(* IEC 61131-3 sources: volt/packages/volt-lsp-iec/test-corpus/lenze-mid/Device/Plc Logic/Application/MotionControl/Lenze, 9 files *)

(* ---- L_GetSlot_i700.pou ---- *)
FUNCTION L_GetSlot_i700 : INT
VAR_IN_OUT
	Axis: AXIS_REF;
END_VAR
VAR
	pAxisRef_i700: POINTER TO _AXIS_REF_i700;
END_VAR

%LANGUAGE ST
//'L_GetSlot_i700'
//
//04.2016
//Lenze Vertrieb GmbH, Mirco Guddat

(***********************************************************************************

This function check if the connected axis is an i700 axis an on witch slot it runs.
Return value:
	0 - No i700 axis
	1 - i700 axis on slot 1
	2 - i700 axis on slot 2

***********************************************************************************)

//Check if this is a i700 axis
IF (Axis.eDeviceOrigin = L_MC1P_DriveType.i700) THEN
	pAxisRef_i700:= ADR(Axis);
	IF pAxisRef_i700^.xSlot2 THEN //Check slot 2
		L_GetSlot_i700:= 2;
	ELSE
		L_GetSlot_i700:= 1;
	END_IF
ELSIF (Axis.eDeviceOrigin = L_MC1P_DriveType.i900) THEN
	L_GetSlot_i700:= 1;
ELSIF (Axis.eDeviceOrigin = L_MC1P_DriveType.i500) THEN
	L_GetSlot_i700:= 1;
ELSE
	L_GetSlot_i700:= 0; //No i700 axis
END_IF

END_FUNCTION

(* ---- ATD_FQI.pou ---- *)
FUNCTION_BLOCK ATD_FQI
VAR_INPUT
	lrAcc: LREAL:=1600;
	lrDec: LREAL:=1600;

END_VAR
VAR_OUTPUT
END_VAR
VAR
	BasicSpeed: L_MC1P_BasicActuatingSpeed;
	OffDelay: TOF;
END_VAR
VAR_IN_OUT
	ioAxis: AXIS_REF;
	DataIO: sUDT_FQIComm_Drive;;
END_VAR
%LANGUAGE LD
%NETWORK "Return when virtual axis"
ASSIGN(ioAxis.xVirtual, Q => RETURN);
%NETWORK
BasicSpeed(Axis := ioAxis, xEnableInternalControl := TRUE, xRegulatorOn := OffDelay(IN := DataIO.Controlword.Bit4_RunForward, PT := T#1S), xResetError := DataIO.Controlword.Bit7_ResetFault, xSetDriveQsp := DataIO.Controlword.Bit2_QuickStop, xEnableSetVel := DataIO.Controlword.Bit4_RunForward, xInvertDirection := DataIO.Controlword.Bit12_ReverseDirection, lrSetVel := DataIO.RefSpeed, lrSetAcc := lrAcc, lrSetDec := lrDec, xAxisReady => DataIO.Status.Bit0_ReadyForOperation, xDriveError => DataIO.Status.Bit3_Fault);

END_FUNCTION_BLOCK

(* ---- ATD_TorqueControl.pou ---- *)
FUNCTION_BLOCK ATD_TorqueControl EXTENDS ATD_FQI
VAR_INPUT
	lrTorque	: LREAL;
END_VAR
VAR_OUTPUT
END_VAR
VAR
	L_MC1P_CyclicParameterAccessWrite_0: L_MC1P_CyclicParameterAccessWrite;
END_VAR

%LANGUAGE LD
%NETWORK
SUPER^(ioAxis := ioAxis, DataIO := DataIO);
%NETWORK
L_MC1P_CyclicParameterAccessWrite_0(Axis := ioAxis, xEnable := TRUE, wIndex := 16#4008, usiSubIndex := 5, usiSize := 2, xSigned := 1, lrScaleFactor := 1, lrData := lrTorque);

END_FUNCTION_BLOCK

(* ---- BasicMovement.pou ---- *)
FUNCTION_BLOCK BasicMovement
//Dataexchange CONTROL ===========
VAR_IN_OUT
	ioDataExchange					:  sUDT_BasicMovementComm_Drive;
END_VAR
VAR_INPUT
	TouchProbeSensor				: BOOL;
	i_lrWindowStandstill			: LREAL;
	i_lrJogVel						: LREAL;
END_VAR
VAR_OUTPUT
END_VAR
VAR
	//ControlWord
	internalControl					:	BOOL;
	Control_Local			 		:	sUDT_BasicMovementComm_Drive_Control;			//output to plc

	//StatusWord

	//instance
	AxisControl						: L_TB2P_BasicMotionBase;
	SetTorqueError					: L_IE1P_SetErrorSingle;
END_VAR
VAR_IN_OUT
	ioSlaveAxis						: AXIS_REF;
END_VAR

%LANGUAGE ST

ReadInputs();
BasicMotionParameters();
BasicMotion();
SetTorqueLimits();
BrakeLogic();
WriteOutputs();

END_FUNCTION_BLOCK

METHOD BasicMotion
VAR_INPUT
END_VAR
VAR_INST
	intPositioningState		: INT;
	R_TRIG_TP				: R_TRIG;
	SetIntQspRamp			: L_SetIntQspRamp;
	lrDecErrorStopOld		: LREAL;
END_VAR
VAR

END_VAR
%LANGUAGE ST

R_TRIG_TP(CLK:=TouchProbeSensor , Q=> );

CASE intPositioningState OF
	0:	(* Wait for synchronisation *)
		AxisControl.scCtrlBasicMotion.xMoveAbsExecute := FALSE;
		AxisControl.scCtrlBasicMotion.xMoveRelExecute := FALSE;
		AxisControl.scCtrlBasicMotion.xMoveVelExecute := FALSE;
		AxisControl.scCtrlBasicMotion.xHalt := FALSE;

		IF Control_Local.StartAbsPos THEN
			intPositioningState:=10;
		ELSIF Control_Local.StartRelPos THEN
			intPositioningState:=20;
		ELSIF Control_Local.StartVelocity THEN
			intPositioningState:=30;
		ELSIF Control_Local.StartTouchprobePos THEN
			intPositioningState:=40;
		ELSIF Control_Local.StartTorqueMode THEN
			intPositioningState:=50;
		END_IF

///////////////////////////////////////////////////////////////////////////
///////////////////////////////Move absolute///////////////////////////////
///////////////////////////////////////////////////////////////////////////

	10:	(*Move absolute to position*)
		AxisControl.scPar.lrAcc := Control_Local.AccUnit;
		AxisControl.scPar.lrDec := Control_Local.DecUnit;
		AxisControl.scPar.lrVel  := Control_Local.VelUnit;
		AxisControl.scCtrlBasicMotion.lrPos_Dist := Control_Local.PosUnit;

		AxisControl.scCtrlBasicMotion.xMoveAbsExecute := TRUE;

		IF AxisControl.scStatusBasicMotion.xFunDone THEN
			ioDataExchange.Status.InPosition:=TRUE;
			intPositioningState:=15;
		ELSIF NOT Control_Local.StartAbsPos THEN
			intPositioningState:=100;
		END_IF

	15:	IF NOT Control_Local.StartAbsPos THEN
			ioDataExchange.Status.InPosition:=FALSE;
			intPositioningState:=0;
		END_IF

///////////////////////////////////////////////////////////////////////////
/////////////////////////////Move Touchprobe///////////////////////////////
///////////////////////////////////////////////////////////////////////////
	40:	(*Move Touchprobe*)
		AxisControl.scPar.lrAcc := Control_Local.AccUnit;
		AxisControl.scPar.lrDec := Control_Local.DecUnit;
		AxisControl.scPar.lrVel := Control_Local.VelUnit;

		AxisControl.scCtrlBasicMotion.xMoveVelExecute := TRUE;

		IF R_TRIG_TP.Q THEN
			AxisControl.scCtrlBasicMotion.lrPos_Dist := Control_Local.PosUnit;
			AxisControl.scCtrlBasicMotion.xMoveRelExecute := TRUE;
			intPositioningState:=41;
		ELSIF NOT Control_Local.StartTouchprobePos THEN
			intPositioningState:=100;
		END_IF

	41://wait for positioning done
		IF AxisControl.scStatusBasicMotion.xFunDone THEN
			ioDataExchange.Status.InPosition:=TRUE;
			intPositioningState:=45;
		ELSIF NOT Control_Local.StartTouchprobePos THEN
			intPositioningState:=100;
		END_IF

	45:	IF NOT Control_Local.StartTouchprobePos THEN
			ioDataExchange.Status.InPosition:=FALSE;
			intPositioningState:=0;
		END_IF

///////////////////////////////////////////////////////////////////////////
///////////////////////////////Stop movement///////////////////////////////
///////////////////////////////////////////////////////////////////////////
	100:(*Stop absolute movement*)
		AxisControl.scCtrlBasicMotion.xHalt := TRUE;

		IF AxisControl.scStatusBasicMotion.xStandstillSetVelocity THEN
			intPositioningState:=0;
		END_IF

END_CASE;

//R_TRIG_TP(CLK:=TouchProbeSensor , Q=> );

AxisControl.scCtrlBasicMotion.xResetHomePosition:=Control_Local.ResetHomePos;

AxisControl(
	xEnable:= TRUE,
	xEnableOperation:=Control_Local.Enable ,
	xResetError:=Control_Local.ResetError ,
	xQSPApplication:= ,
	xAbort:= ,
	xJogPos:= ,
	xJogNeg:= ,
	xHomeExecute:= Control_Local.ActivateHoming,
	lrOverride:= ,
	scCtrlBasicMotion:= ,
	scPar:= ,
	Axis:=ioSlaveAxis ,
	xReadyForOperation=> ,
	xOperationEnabled=> ,
	xReadyForMotion=> ,
	xError=> ,
	xWarning=> ,
	eErrorID=> ,
	xSTOActive=> ,
	xQSPActive=> ,
	xAbortBusy=> ,
	xAbortDone=> ,
	xJoggingBusy=> ,
	xHomingBusy=> ,
	xHomingDone=> ,
	xIsHomed=> ,
	eTMState=> ,
	scStatusBasicMotion=> ,
	lrActVel=> ,
	lrSetVelOut=> ,
	lrActPos=> ,
	lrSetPosOut=> ,
	lrActFollowingError=> );

SetIntQspRamp(
	Axis:=ioSlaveAxis ,
	xExecute:=ioSlaveAxis.xAxisAvailable AND NOT ioSlaveAxis.xVirtual AND (lrDecErrorStopOld=ioSlaveAxis.lrDecErrorStop) ,
	lrQspRamp:=ioSlaveAxis.lrDecErrorStop ,
	lrQspTime:= ,
	xUseQspTime:= ,
	xBusy=> ,
	xDone=> ,
	xError=> ,
	eErrorID=> );
lrDecErrorStopOld:=ioSlaveAxis.lrDecErrorStop;
END_METHOD

METHOD BasicMotionParameters
VAR_INPUT
END_VAR

%LANGUAGE ST
//General
//ioSlaveAxis.scPar.WindowStandStill:=i_lrWindowStandstill;
//ioSlaveAxis.scPar.JoggingSetVel:=i_lrJogVel;
//ioSlaveAxis.scPar.JoggingSetAcc:=i_lrJogVel*10;
//ioSlaveAxis.scPar.JoggingSetDec:=i_lrJogVel*10;
//ioSlaveAxis.scPar.JoggingSetJerk:=0;
END_METHOD

METHOD BrakeLogic
VAR_INPUT

END_VAR
VAR_INST
	BrakeInterface			: L_MC1P_BrakeInterface;
END_VAR

VAR

END_VAR
%LANGUAGE ST

BrakeInterface(
	Axis:= ioSlaveAxis,
	xEnable:= NOT ioSlaveAxis.xVirtual ,
	xReleaseBrake:= Control_Local.ReleaseBrake,
	lrTorqueAdd:= ,
	xBrakeModeActivate:= ,
	eBrakeMode:= ,
	xValid=> ,
	xBusy=> ,
	xError=> ,
	eErrorID=> ,
	xBrakeReleaseOut=> ,
	xBrakeReleased=> ,
	lrActTorque=> ,
	lrStartingTorqueSaved=> ,
	lrStartingTorqueEffective=> ,
	eBrakeModeActive=> );
END_METHOD

METHOD ReadInputs
VAR_INPUT
END_VAR

%LANGUAGE ST

//activate internal control
IF NOT internalControl THEN
	Control_Local	:= ioDataExchange.Control;
END_IF

END_METHOD

METHOD SetTorqueLimits
VAR_INPUT

END_VAR
VAR_INST
	TorqueLimit						: L_MC1P_SetTorqueLimit;
	lrRefTorqueAxis					: LREAL;
	lrActTorqueProcent				: LREAL;
	ResetError						: L_IE1P_ResetError;
END_VAR

VAR

END_VAR
%LANGUAGE ST

//Max torque on the axis. If the machine doesn't stop due to a programming error, this part ensures that the torque never gets too high.
TorqueLimit(
	Axis:= ioSlaveAxis,
	xEnable:= NOT ioSlaveAxis.xVirtual ,
	xSetTorqueLimitPos:= TRUE,
	lrTorqueLimitPos:= (Control_Local.TorqueLimit/100)*1.1, 				//The max torque allowed on the axis is 10% higher then the alarm value.
	xSetTorqueLimitNeg:= TRUE,
	lrTorqueLimitNeg:= (Control_Local.TorqueLimit/100)*1.1, 				//The max torque allowed on the axis is 10% higher then the alarm value.
	xTorqueInputAsPercent:= TRUE,
	xBusy=> ,
	xError=> ,
	eErrorID=> );

lrRefTorqueAxis := L_MC1P_GetRatedTorqueAxis(Axis:=ioSlaveAxis);
//Torque limit error
IF lrRefTorqueAxis > 0 THEN
	lrActTorqueProcent := ABS(ioSlaveAxis.lrActTorque/lrRefTorqueAxis);
END_IF

SetTorqueError(
	ModuleHandler:= ,
	ErrorHandler:=ioSlaveAxis ,
	xSetError:=lrActTorqueProcent > (Control_Local.TorqueLimit/100) ,
	eSeverity:=L_IE1P_SeverityLevel.Fault_QspAppl ,
	wTextRefId:= ATD_Errorlist,
	wErrorId:= 1,
	eReaction:= ,
	eGroup:= ,
	xError=> ,
	eErrorID=> ,
	scErrorInformation=> );

ResetError(
	ModuleHandler:= ,
	ErrorHandler:=ioSlaveAxis ,
	xResetError:=AxisControl.xResetError ,
	xError=> ,
	eErrorID=> ,
	xErrorResetActive=> ,
	xResetActive=> );
END_METHOD

METHOD WriteOutputs
VAR_INPUT
END_VAR
VAR_INST

END_VAR

%LANGUAGE ST

ioDataExchange.Status.DriveCommAlive				:= ioSlaveAxis.xCommunicationOK;
ioDataExchange.Status.ReadyForOperation				:= AxisControl.xReadyForOperation;
ioDataExchange.Status.ReadyForMotion				:= AxisControl.xReadyForMotion;
ioDataExchange.Status.HomingPosOK					:= AxisControl.xIsHomed;
ioDataExchange.Status.InPosition					;//writen in statemachine
ioDataExchange.Status.VelocitySetpointReached		;//writen in statemachine
ioDataExchange.Status.ActSpeed						:= AxisControl.lrActVel;
ioDataExchange.Status.ActPos						:= AxisControl.lrActPos;

END_METHOD

(* ---- Camming.pou ---- *)
FUNCTION_BLOCK Camming
//Dataexchange CONTROL ===========
VAR_IN_OUT
	ioDataExchange					:  sUDT_ServoComm_Drive;
END_VAR
VAR_INPUT

	i_xOnlyPositiveDirectionSync	: BOOL;
	i_lrWindowStandstill			: LREAL;
	i_lrJogVel						: LREAL;
	i_lrSyncVel 					: LREAL;
	i_NormalCamRefTable				: MC_CAM_REF;
	i_ByPassCamRefTable				: MC_CAM_REF;
	i_CamCyclic						: BOOL;
	i_MasterAbsolute				: BOOL;
	i_SlaveAbsolute					: BOOL;
END_VAR
VAR
	//ControlWord
	internalControl					:	BOOL;
	Control_Local			 		:	sUDT_ServoComm_Drive_Control;			//output to plc

	//StatusWord

	//instance
	AxisControl						: L_TS2P_FlexCamState;
	SetTorqueError					: L_IE1P_SetErrorSingle;
END_VAR
VAR_IN_OUT
	ioMasterAxis					: AXIS_REF;
	ioSlaveAxis						: AXIS_REF;
END_VAR

%LANGUAGE ST

ReadInputs();
FlexCamParameters();
FlexCam();
SetTorqueLimits();
BrakeLogic();
WriteOutputs();

END_FUNCTION_BLOCK

METHOD BrakeLogic
VAR_INPUT

END_VAR
VAR_INST
	BrakeInterface			: L_MC1P_BrakeInterface;
END_VAR

VAR

END_VAR
%LANGUAGE ST

BrakeInterface(
	Axis:= ioSlaveAxis,
	xEnable:= NOT ioSlaveAxis.xVirtual ,
	xReleaseBrake:= Control_Local.ReleaseBrake,
	lrTorqueAdd:= ,
	xBrakeModeActivate:= ,
	eBrakeMode:= ,
	xValid=> ,
	xBusy=> ,
	xError=> ,
	eErrorID=> ,
	xBrakeReleaseOut=> ,
	xBrakeReleased=> ,
	lrActTorque=> ,
	lrStartingTorqueSaved=> ,
	lrStartingTorqueEffective=> ,
	eBrakeModeActive=> );
END_METHOD

METHOD FlexCam
VAR_INPUT
END_VAR

VAR_INST
	lrMasterPos				: LREAL;
	lrSlavePos				: LREAL;
	lrDifferenceCalc		: LREAL;
	intSyncState			: INT;

	uiSetCamTable			: UINT;
	itfActiveCamTable		: MC_CAM_REF;
	CamGetSlavePosition		: L_MC2P_CamGetSlavePosition;
	xSyncCam				: BOOL;
	DelayHomePosReset	: TON;

	SetIntQspRamp			: L_SetIntQspRamp;
	lrDecErrorStopOld		: LREAL;
END_VAR
VAR

END_VAR
%LANGUAGE ST
//Selection of the cam.
IF Control_Local.SelectBypassCAM THEN
	uiSetCamTable := 2;					//Camtable 2 is a zero curve.
	itfActiveCamTable := i_ByPassCamRefTable;
ELSE
	uiSetCamTable := 1;					//Camtable 1 is the normal curve.
	itfActiveCamTable := i_NormalCamRefTable;
END_IF

//Settings for only positive synchronisation direction
IF i_xOnlyPositiveDirectionSync = TRUE AND i_SlaveAbsolute THEN

	//Get master position
	lrMasterPos := ((ioMasterAxis.lrSetPosition * AxisControl.lrSetScalingX) + AxisControl.lrSetOffsetPosX);
	IF ioMasterAxis.eTraversingRange = L_MC1P_TRAVERSINGRANGE.Modulo THEN
		lrMasterPos := L_MC1P_ModuloCycle(lrMasterPos, ioMasterAxis.lrCycleLength);
	END_IF

	//Get slave position
	CamGetSlavePosition(
		xExecute:= Control_Local.ActivateCamming,
		lrMasterPosition:= lrMasterPos,
		itfCamTable:= itfActiveCamTable,
		xDone=> ,
		xBusy=> ,
		xError=> ,
		eErrorID=> ,
		lrSlavePosition=> );
	lrSlavePos := ((CamGetSlavePosition.lrSlavePosition * AxisControl.lrSetScalingY) + AxisControl.lrSetOffsetPosY);
	IF ioSlaveAxis.eTraversingRange = L_MC1P_TRAVERSINGRANGE.Modulo THEN
		lrSlavePos := L_MC1P_ModuloCycle(lrSlavePos, ioSlaveAxis.lrCycleLength);
	END_IF

	//Calculate position difference between master and slave
	lrDifferenceCalc := L_MC1P_HlpModuloDiff(
					lrDiff:= (ioSlaveAxis.lrSetPosition - lrSlavePos),
					lrLen := ioSlaveAxis.lrCycleLength);

	//Start synchronisation
	IF ABS(lrDifferenceCalc) < 0.2 THEN
		AxisControl.scPar.eDirection := MC_DIRECTION.mcShortestWay;
	ELSE
		AxisControl.scPar.eDirection := MC_DIRECTION.mcPositiveDirection;
	END_IF

	IF NOT AxisControl.xReadyForMotion AND intSyncState>0 THEN
		intSyncState:=0;
	END_IF

	CASE intSyncState OF
		0:	(* Wait for synchronisation *)
			xSyncCam := FALSE;
			AxisControl.scCtrlBasicMotion.xMoveAbsExecute := FALSE;
			AxisControl.scCtrlBasicMotion.xHalt:=FALSE;
			AxisControl.xQSPApplication:=FALSE;

			IF Control_Local.ActivateCamming AND AxisControl.xReadyForMotion THEN
				intSyncState := 1;
			END_IF

		1:	(*Move absolute to position*)
			AxisControl.scCtrlBasicMotion.lrPos_Dist := lrSlavePos;
			AxisControl.scPar.lrAcc := AxisControl.scPar.lrSyncAcc;
			AxisControl.scPar.lrDec := AxisControl.scPar.lrSyncDec;
			AxisControl.scPar.lrVel  := AxisControl.scPar.lrSyncVel;

			AxisControl.scCtrlBasicMotion.xMoveAbsExecute := Control_Local.ActivateCamming AND CamGetSlavePosition.xDone;

			IF Control_Local.ActivateCamming = FALSE THEN
				intSyncState := 2;
			ELSIF AxisControl.scStatusBasicMotion.xFunDone = TRUE THEN
				intSyncState := 3;
			END_IF

		2:	(*Stop absolute movement*)
			AxisControl.scCtrlBasicMotion.xMoveAbsExecute := FALSE;
			AxisControl.scCtrlBasicMotion.xHalt:=TRUE;

			IF AxisControl.scStatusBasicMotion.xFunDone = TRUE THEN
				intSyncState := 0;
			END_IF

		3:	(*Synchronise drive*)
			xSyncCam := TRUE;

			IF Control_Local.ActivateCamming = FALSE THEN
				AxisControl.xQSPApplication:=TRUE;
				intSyncState := 4;
			END_IF

		4:	IF ioSlaveAxis.xStandstillSetVelocity THEN
				AxisControl.xQSPApplication:=FALSE;
				intSyncState := 0;
			END_IF

	END_CASE;
ELSE
	xSyncCam := Control_Local.ActivateCamming;
END_IF

AxisControl.scCtrlBasicMotion.xResetHomePosition:=Control_Local.ResetHomePos;

 DelayHomePosReset(IN:= NOT AxisControl.xIsHomed, PT:=T#10MS);

AxisControl(
	xEnable:=TRUE ,
	xEnableOperation:= Control_Local.Enable,
	xResetError:= Control_Local.ResetError,
	xQSPApplication:=  ,
	xAbort:=,
	xJogPos:= ,
	xJogNeg:= ,
	xHomeExecute:= Control_Local.SetHomePos AND DelayHomePosReset.q,
	lrOverride:= ,
	scCtrlBasicMotion:= ,
	scPar:= ,
	Axis:= ioSlaveAxis,
	scAccessPoints:= ,
	MasterValues:= ioMasterAxis,
	xSyncIn:= xSyncCam ,
	xCamChangeInstant:= ,
	lrSetOffsetPosX:= Control_Local.XOffset,
	lrSetOffsetPosY:= Control_Local.YOffset,
	lrSetScalingX:= ,
	lrSetScalingY:= Control_Local.YScale/1000,
	CamTable1:= i_NormalCamRefTable,
	CamTable2:= i_ByPassCamRefTable,
	CamTable3:= ,
	CamTable4:= ,
	wSetCamTable:= uiSetCamTable,
	xCamSequencer:= ,
	xReadyForOperation=> ,
	xOperationEnabled=> ,
	xReadyForMotion=> ,
	xError=> ,
	xWarning=> ,
	eErrorID=>  ,
	xSTOActive=> ,
	xQSPActive=> ,
	xAbortBusy=> ,
	xAbortDone=> ,
	xJoggingBusy=> ,
	xHomingBusy=> ,
	xHomingDone=> ,
	xIsHomed=> ,
	eTMState=> ,
	scStatusBasicMotion=> ,
	lrActVel=> ,
	lrSetVelOut=> ,
	lrActPos=> ,
	lrSetPosOut=> ,
	lrActFollowingError=> ,
	scSignalFlow=> ,
	xSynchronised=> ,
	xAccDecSync=> ,
	xCammingBusy=> ,
	xEndOfProfile=> ,
	lrOffsetPosX=> ,
	lrOffsetPosY=> ,
	wActiveCamTable=> ,
	xCamSequencerActive=> );

SetIntQspRamp(
	Axis:=ioSlaveAxis ,
	xExecute:=ioSlaveAxis.xAxisAvailable AND NOT ioSlaveAxis.xVirtual AND (lrDecErrorStopOld=ioSlaveAxis.lrDecErrorStop) ,
	lrQspRamp:=ioSlaveAxis.lrDecErrorStop ,
	lrQspTime:= ,
	xUseQspTime:= ,
	xBusy=> ,
	xDone=> ,
	xError=> ,
	eErrorID=> );
lrDecErrorStopOld:=ioSlaveAxis.lrDecErrorStop;
END_METHOD

METHOD FlexCamParameters
VAR_INPUT
END_VAR

%LANGUAGE ST
//General
//ioSlaveAxis.scPar.WindowStandStill:=i_lrWindowStandstill;
//ioSlaveAxis.scPar.JoggingSetVel:=i_lrJogVel;
//ioSlaveAxis.scPar.JoggingSetAcc:=i_lrJogVel*10;
//ioSlaveAxis.scPar.JoggingSetDec:=i_lrJogVel*10;
//ioSlaveAxis.scPar.JoggingSetJerk:=0;
//Set Flexcam Parameters
AxisControl.scPar.lrSyncVel:=i_lrSyncVel;
AxisControl.scPar.lrSyncAcc:=i_lrSyncVel*10;
AxisControl.scPar.lrSyncDec:=i_lrSyncVel*10;
AxisControl.scPar.lrSyncJerk:=0;//i_lrSyncVel*100;

AxisControl.scPar.lrSetOffsetScalingXVel:=i_lrSyncVel;
AxisControl.scPar.lrSetOffsetScalingXAcc:=i_lrSyncVel*10;
AxisControl.scPar.lrSetOffsetScalingXDec:=i_lrSyncVel*10;
AxisControl.scPar.lrSetOffsetScalingXJerk:=0;//i_lrSyncVel*100;

AxisControl.scPar.lrSetOffsetScalingYVel:=i_lrSyncVel;
AxisControl.scPar.lrSetOffsetScalingYAcc:=i_lrSyncVel*10;
AxisControl.scPar.lrSetOffsetScalingYDec:=i_lrSyncVel*10;
AxisControl.scPar.lrSetOffsetScalingYJerk:=0;//i_lrSyncVel*100;

AxisControl.scPar.eOffsetModeX:=L_TS2P_OffsetMode.ProfGenAbsolute;
AxisControl.scPar.eOffsetModeY:=L_TS2P_OffsetMode.ProfGenAbsolute;

AxisControl.scPar.eScalingModeX:=L_TS2P_ScalingMode.x_zero;
AxisControl.scPar.eScalingModeY:=L_TS2P_ScalingMode.x_zero;

AxisControl.scPar.xCamCyclic:=i_CamCyclic;
AxisControl.scPar.xMasterAbsolute:=i_MasterAbsolute;
AxisControl.scPar.xSlaveAbsolute:=i_SlaveAbsolute;

IF i_SlaveAbsolute THEN
	AxisControl.scPar.eSyncMode:=L_TS2P_SyncModeFlexCam.ProfGenAbsolute;
ELSE
	AxisControl.scPar.eSyncMode:=L_TS2P_SyncModeFlexCam.InstantRelative;
END_IF
AxisControl.scPar.lrSlaveSyncOutPos:=AxisControl.lrSetPosOut;

END_METHOD

METHOD ReadInputs
VAR_INPUT
END_VAR

%LANGUAGE ST

//activate internal control
IF NOT internalControl THEN
	Control_Local	:= ioDataExchange.Control;
END_IF

END_METHOD

METHOD SetTorqueLimits
VAR_INPUT

END_VAR
VAR_INST
	TorqueLimit						: L_MC1P_SetTorqueLimit;
	lrRefTorqueAxis					: LREAL;
	lrActTorqueProcent				: LREAL;
	ResetError						: L_IE1P_ResetError;
END_VAR

VAR

END_VAR
%LANGUAGE ST

//Max torque on the axis. If the machine doesn't stop due to a programming error, this part ensures that the torque never gets too high.
TorqueLimit(
	Axis:= ioSlaveAxis,
	xEnable:= NOT ioSlaveAxis.xVirtual ,
	xSetTorqueLimitPos:= TRUE,
	lrTorqueLimitPos:= (Control_Local.TorqueLimit/100)*1.1, 				//The max torque allowed on the axis is 10% higher then the alarm value.
	xSetTorqueLimitNeg:= TRUE,
	lrTorqueLimitNeg:= (Control_Local.TorqueLimit/100)*1.1, 				//The max torque allowed on the axis is 10% higher then the alarm value.
	xTorqueInputAsPercent:= TRUE,
	xBusy=> ,
	xError=> ,
	eErrorID=> );

lrRefTorqueAxis := L_MC1P_GetRatedTorqueAxis(Axis:=ioSlaveAxis);
//Torque limit error
IF lrRefTorqueAxis > 0 THEN
	lrActTorqueProcent := ABS(ioSlaveAxis.lrActTorque/lrRefTorqueAxis);
END_IF

SetTorqueError(
	ModuleHandler:= ,
	ErrorHandler:=ioSlaveAxis ,
	xSetError:=lrActTorqueProcent > (Control_Local.TorqueLimit/100) ,
	eSeverity:=L_IE1P_SeverityLevel.Fault_Qsp_Cinh ,
	wTextRefId:= ATD_Errorlist,
	wErrorId:= 1,
	eReaction:= ,
	eGroup:= ,
	xError=> ,
	eErrorID=> ,
	scErrorInformation=> );

ResetError(
	ModuleHandler:= ,
	ErrorHandler:=ioSlaveAxis ,
	xResetError:=AxisControl.xResetError ,
	xError=> ,
	eErrorID=> ,
	xErrorResetActive=> ,
	xResetActive=> );
END_METHOD

METHOD WriteOutputs
VAR_INPUT
END_VAR
VAR_INST

END_VAR

%LANGUAGE ST

ioDataExchange.Status.DriveCommAlive				:= ioSlaveAxis.xCommunicationOK;
ioDataExchange.Status.ReadyForOperation				:= AxisControl.xReadyForOperation;
ioDataExchange.Status.ReadyForMotion				:= AxisControl.xReadyForMotion;
ioDataExchange.Status.HomingPosOK					:= AxisControl.xIsHomed;
ioDataExchange.Status.InSync						:= AxisControl.xSynchronised;
ioDataExchange.Status.TorqueLimit					:= SetTorqueError.scErrorInformation.xError;
ioDataExchange.Status.ActSpeed						:= AxisControl.lrActVel;
ioDataExchange.Status.ActPos						:= AxisControl.lrActPos;

END_METHOD

(* ---- Camming_SideCorrection.pou ---- *)
FUNCTION_BLOCK Camming_SideCorrection EXTENDS Camming
VAR_INPUT
	i_NormalCamRefTableNeg				: MC_CAM_REF;
END_VAR
VAR_OUTPUT
END_VAR
VAR
END_VAR

%LANGUAGE ST
SUPER^( ioDataExchange:=ioDataExchange, ioMasterAxis:=ioMasterAxis,ioSlaveAxis:=ioSlaveAxis);

END_FUNCTION_BLOCK

METHOD FlexCam
VAR_INPUT
END_VAR

VAR_INST
	lrMasterPos				: LREAL;
	lrSlavePos				: LREAL;
	lrDifferenceCalc		: LREAL;
	intSyncState			: INT;

	uiSetCamTable			: UINT;
	itfActiveCamTable		: MC_CAM_REF;
	CamGetSlavePosition		: L_MC2P_CamGetSlavePosition;
	xSyncCam				: BOOL;

END_VAR
VAR

END_VAR
%LANGUAGE ST
//Selection of the cam.
IF Control_Local.SelectBypassCAM THEN
	uiSetCamTable := 2;					//Camtable 2 is a zero curve.
ELSE
	IF Control_Local.YScale<0 THEN
		uiSetCamTable := 3;					//Camtable 1 is the normal curve.
	ELSE
		uiSetCamTable := 1;					//Camtable 1 is the normal curve.
	END_IF
END_IF

//Settings for only positive synchronisation direction
IF i_xOnlyPositiveDirectionSync = TRUE AND i_SlaveAbsolute THEN

	//Get master position
	lrMasterPos := ((ioMasterAxis.lrSetPosition * AxisControl.lrSetScalingX) + AxisControl.lrSetOffsetPosX);
	IF ioMasterAxis.eTraversingRange = L_MC1P_TRAVERSINGRANGE.Modulo THEN
		lrMasterPos := L_MC1P_ModuloCycle(lrMasterPos, ioMasterAxis.lrCycleLength);
	END_IF

	//Get slave position
	CamGetSlavePosition(
		xExecute:= Control_Local.ActivateCamming,
		lrMasterPosition:= lrMasterPos,
		itfCamTable:= itfActiveCamTable,
		xDone=> ,
		xBusy=> ,
		xError=> ,
		eErrorID=> ,
		lrSlavePosition=> );
	lrSlavePos := ((CamGetSlavePosition.lrSlavePosition * AxisControl.lrSetScalingY) + AxisControl.lrSetOffsetPosY);
	IF ioSlaveAxis.eTraversingRange = L_MC1P_TRAVERSINGRANGE.Modulo THEN
		lrSlavePos := L_MC1P_ModuloCycle(lrSlavePos, ioSlaveAxis.lrCycleLength);
	END_IF

	//Calculate position difference between master and slave
	lrDifferenceCalc := L_MC1P_HlpModuloDiff(
					lrDiff:= (ioSlaveAxis.lrSetPosition - lrSlavePos),
					lrLen := ioSlaveAxis.lrCycleLength);

	//Start synchronisation
	IF ABS(lrDifferenceCalc) < 0.2 THEN
		AxisControl.scPar.eDirection := MC_DIRECTION.mcShortestWay;
	ELSE
		AxisControl.scPar.eDirection := MC_DIRECTION.mcPositiveDirection;
	END_IF

	IF NOT AxisControl.xReadyForMotion AND intSyncState>0 THEN
		intSyncState:=0;
	END_IF

	CASE intSyncState OF
		0:	(* Wait for synchronisation *)
			xSyncCam := FALSE;
			AxisControl.scCtrlBasicMotion.xMoveAbsExecute := FALSE;
			AxisControl.scCtrlBasicMotion.xHalt:=FALSE;

			IF Control_Local.ActivateCamming AND AxisControl.xReadyForMotion THEN
				intSyncState := 1;
			END_IF

		1:	(*Move absolute to position*)
			AxisControl.scCtrlBasicMotion.lrPos_Dist := lrSlavePos;
			AxisControl.scPar.lrAcc := AxisControl.scPar.lrSyncAcc;
			AxisControl.scPar.lrDec := AxisControl.scPar.lrSyncDec;
			AxisControl.scPar.lrVel  := AxisControl.scPar.lrSyncVel;

			AxisControl.scCtrlBasicMotion.xMoveAbsExecute := Control_Local.ActivateCamming AND CamGetSlavePosition.xDone;

			IF Control_Local.ActivateCamming = FALSE THEN
				intSyncState := 2;
			ELSIF AxisControl.scStatusBasicMotion.xFunDone = TRUE THEN
				intSyncState := 3;
			END_IF

		2:	(*Stop absolute movement*)
			AxisControl.scCtrlBasicMotion.xMoveAbsExecute := FALSE;
			AxisControl.scCtrlBasicMotion.xHalt:=TRUE;

			IF AxisControl.scStatusBasicMotion.xFunDone = TRUE THEN
				intSyncState := 0;
			END_IF

		3:	(*Synchronise drive*)
			xSyncCam := TRUE;

			IF Control_Local.ActivateCamming = FALSE THEN
				intSyncState := 0;
			END_IF

	END_CASE;
ELSE
	xSyncCam := Control_Local.ActivateCamming;
END_IF

AxisControl.scCtrlBasicMotion.xResetHomePosition:=Control_Local.ResetHomePos;

AxisControl(
	xEnable:=TRUE ,
	xEnableOperation:= Control_Local.Enable,
	xResetError:= Control_Local.ResetError,
	xQSPApplication:= ,
	xAbort:= ,
	xJogPos:= Control_Local.Spare2,
	xJogNeg:= Control_Local.Spare1,
	xHomeExecute:= Control_Local.SetHomePos,
	lrOverride:= ,
	scCtrlBasicMotion:= ,
	scPar:= ,
	Axis:= ioSlaveAxis,
	scAccessPoints:= ,
	MasterValues:= ioMasterAxis,
	xSyncIn:= xSyncCam,
	xCamChangeInstant:= ,
	lrSetOffsetPosX:= Control_Local.XOffset,
	lrSetOffsetPosY:= Control_Local.YOffset,
	lrSetScalingX:= ,
	lrSetScalingY:= ABS(Control_Local.YScale/1000),
	CamTable1:= i_NormalCamRefTable,
	CamTable2:= i_ByPassCamRefTable,
	CamTable3:= i_NormalCamRefTableNeg ,
	CamTable4:= ,
	wSetCamTable:= uiSetCamTable,
	xCamSequencer:= ,
	xReadyForOperation=> ,
	xOperationEnabled=> ,
	xReadyForMotion=> ,
	xError=> ,
	xWarning=> ,
	eErrorID=>  ,
	xSTOActive=> ,
	xQSPActive=> ,
	xAbortBusy=> ,
	xAbortDone=> ,
	xJoggingBusy=> ,
	xHomingBusy=> ,
	xHomingDone=> ,
	xIsHomed=> ,
	eTMState=> ,
	scStatusBasicMotion=> ,
	lrActVel=> ,
	lrSetVelOut=> ,
	lrActPos=> ,
	lrSetPosOut=> ,
	lrActFollowingError=> ,
	scSignalFlow=> ,
	xSynchronised=> ,
	xAccDecSync=> ,
	xCammingBusy=> ,
	xEndOfProfile=> ,
	lrOffsetPosX=> ,
	lrOffsetPosY=> ,
	wActiveCamTable=> ,
	xCamSequencerActive=> );
END_METHOD

(* ---- identPolePosition.pou ---- *)
FUNCTION_BLOCK identPolePosition
VAR_INPUT
	execute				: BOOL;
END_VAR
VAR_OUTPUT
	busy				: BOOL;
	done				: BOOL;
	doneOnce			: BOOL;
	error				: BOOL;
	polePositionOld		: LREAL;
	polePositionNew		: LREAL;
END_VAR
VAR
	iStep: INT;
	MC_ReadParameter	: MC_ReadParameter;
	MC_WriteParameter	: MC_WriteParameter;
	TON:TON;
END_VAR
VAR_IN_OUT
	ioAxis				: AXIS_REF;
END_VAR
%LANGUAGE ST

CASE iStep OF

	0:	MC_ReadParameter.Enable:=FALSE;
		MC_WriteParameter.Execute:=FALSE;
		done:=FALSE;
		busy:=FALSE;
		error:=FALSE;

		IF execute THEN
			busy:=true;
			iStep:=2;
		END_IF

	2:	//Read	0x3024:0	Device control via PDO: Activation	Activate [1]
		MC_ReadParameter.Enable:=TRUE;
		MC_ReadParameter.ParameterNumber:=L_MC1P_IndexToParameter2(
				uiIndex:=16#3024 ,
				usiSubIndex:=0 ,
				uiByteLength:=1 ,
				xUnsigned:=TRUE );

		IF MC_ReadParameter.Valid THEN
			//IF MC_ReadParameter.Value = 1 THEN
				MC_ReadParameter.Enable:=FALSE;
				iStep:=4;
			//ELSE
			//	error:=TRUE;
			//END_IF
		ELSIF NOT execute THEN
			iStep:=0;
		ELSIF MC_ReadParameter.Error THEN
			error:=TRUE;
		END_IF

	4:	//Write	0x3024:0	Device control via PDO: Activation	Off [0]
		MC_WriteParameter.Execute:=TRUE;
		MC_WriteParameter.ParameterNumber:=L_MC1P_IndexToParameter2(
				uiIndex:=16#3024 ,
				usiSubIndex:=0 ,
				uiByteLength:=1 ,
				xUnsigned:=TRUE );
		MC_WriteParameter.Value:=0;

		IF MC_WriteParameter.Done THEN
			MC_WriteParameter.Execute:=FALSE;
			iStep:=6;
		ELSIF NOT execute THEN
			iStep:=0;
		ELSIF MC_WriteParameter.Error THEN
			error:=TRUE;
		END_IF

	6:	//Read	0x3025:0	Mode: Selection	CiA402 mode active [0]
		MC_ReadParameter.Enable:=TRUE;
		MC_ReadParameter.ParameterNumber:=L_MC1P_IndexToParameter2(
				uiIndex:=16#3025 ,
				usiSubIndex:=0 ,
				uiByteLength:=1 ,
				xUnsigned:=TRUE );

		IF MC_ReadParameter.Valid THEN
			//IF MC_ReadParameter.Value = 0 THEN
				MC_ReadParameter.Enable:=FALSE;
				iStep:=8;
			//ELSE
			//	error:=TRUE;
			//END_IF
		ELSIF NOT execute THEN
			iStep:=0;
		ELSIF MC_ReadParameter.Error THEN
			error:=TRUE;
		END_IF

	8:	//Write	0x3025:0	Mode: Selection	Pole position identification PPI (without movement) [7]
		MC_WriteParameter.Execute:=TRUE;
		MC_WriteParameter.ParameterNumber:=L_MC1P_IndexToParameter2(
				uiIndex:=16#3025 ,
				usiSubIndex:=0 ,
				uiByteLength:=1 ,
				xUnsigned:=TRUE );
		MC_WriteParameter.Value:=7;

		IF MC_WriteParameter.Done THEN
			MC_WriteParameter.Execute:=FALSE;
			iStep:=10;
		ELSIF NOT execute THEN
			iStep:=0;
		ELSIF MC_WriteParameter.Error THEN
			error:=TRUE;
		END_IF

	10:	//Read	0x3403:4	Motor (SM): Pole position encoder	49,5	°
		MC_ReadParameter.Enable:=TRUE;
		MC_ReadParameter.ParameterNumber:=L_MC1P_IndexToParameter2(
				uiIndex:=16#3403 ,
				usiSubIndex:=4 ,
				uiByteLength:=2 ,
				xUnsigned:=TRUE );

		IF MC_ReadParameter.Valid THEN
			polePositionOld:=MC_ReadParameter.Value;
			MC_ReadParameter.Enable:=FALSE;
			iStep:=12;
		ELSIF NOT execute THEN
			iStep:=0;
		ELSIF MC_ReadParameter.Error THEN
			error:=TRUE;
		END_IF

	12://Write	0x6840:0	Controlword	0x0006
		MC_WriteParameter.Execute:=TRUE;
		MC_WriteParameter.ParameterNumber:=L_MC1P_IndexToParameter2(
				uiIndex:=16#6840 ,
				usiSubIndex:=0 ,
				uiByteLength:=2 ,
				xUnsigned:=TRUE );
		MC_WriteParameter.Value:=16#0006;

		IF MC_WriteParameter.Done THEN
			MC_WriteParameter.Execute:=FALSE;
			iStep:=14;
		ELSIF NOT execute THEN
			iStep:=0;
		ELSIF MC_WriteParameter.Error THEN
			error:=TRUE;
		END_IF

	14://Read	0x6841:0	Statusword	0x0021
		MC_ReadParameter.Enable:=TRUE;
		MC_ReadParameter.ParameterNumber:=L_MC1P_IndexToParameter2(
				uiIndex:=16#6841 ,
				usiSubIndex:=0 ,
				uiByteLength:=2 ,
				xUnsigned:=TRUE );

		IF MC_ReadParameter.Valid THEN
			//IF MC_ReadParameter.Value = 16#0021 THEN
				MC_ReadParameter.Enable:=FALSE;
				iStep:=16;
			//ELSE
			//	error:=TRUE;
			//END_IF
		ELSIF NOT execute THEN
			iStep:=0;
		ELSIF MC_ReadParameter.Error THEN
			error:=TRUE;
		END_IF

	16://Write	0x6840:0	Controlword	0x0007
		MC_WriteParameter.Execute:=TRUE;
		MC_WriteParameter.ParameterNumber:=L_MC1P_IndexToParameter2(
				uiIndex:=16#6840 ,
				usiSubIndex:=0 ,
				uiByteLength:=2 ,
				xUnsigned:=TRUE );
		MC_WriteParameter.Value:=16#0007;

		IF MC_WriteParameter.Done THEN
			MC_WriteParameter.Execute:=FALSE;
			iStep:=18;
		ELSIF NOT execute THEN
			iStep:=0;
		ELSIF MC_WriteParameter.Error THEN
			error:=TRUE;
		END_IF

	18://Read	0x6841:0	Statusword	0x0023
		MC_ReadParameter.Enable:=TRUE;
		MC_ReadParameter.ParameterNumber:=L_MC1P_IndexToParameter2(
				uiIndex:=16#6841 ,
				usiSubIndex:=0 ,
				uiByteLength:=2 ,
				xUnsigned:=TRUE );

		IF MC_ReadParameter.Valid THEN
			//IF MC_ReadParameter.Value = 16#0023 THEN
				MC_ReadParameter.Enable:=FALSE;
				iStep:=20;
			//ELSE
			//	error:=TRUE;
			//END_IF
		ELSIF NOT execute THEN
			iStep:=0;
		ELSIF MC_ReadParameter.Error THEN
			error:=TRUE;
		END_IF

	20://Write	0x6840:0	Controlword	0x000F
		MC_WriteParameter.Execute:=TRUE;
		MC_WriteParameter.ParameterNumber:=L_MC1P_IndexToParameter2(
				uiIndex:=16#6840 ,
				usiSubIndex:=0 ,
				uiByteLength:=2 ,
				xUnsigned:=TRUE );
		MC_WriteParameter.Value:=16#000F;

		IF MC_WriteParameter.Done THEN
			MC_WriteParameter.Execute:=FALSE;
			TON(IN:=FALSE);
			iStep:=22;
		ELSIF NOT execute THEN
			iStep:=0;
		ELSIF MC_WriteParameter.Error THEN
			error:=TRUE;
		END_IF

	22://Check for finished
		TON(IN:=TRUE , PT:= T#5S, Q=> , ET=> );

		IF TON.Q THEN
			iStep:=24;
		ELSIF NOT execute THEN
			iStep:=0;
		END_IF

	24://Write	0x6840:0	Controlword	0x0000
		MC_WriteParameter.Execute:=TRUE;
		MC_WriteParameter.ParameterNumber:=L_MC1P_IndexToParameter2(
				uiIndex:=16#6840 ,
				usiSubIndex:=0 ,
				uiByteLength:=2 ,
				xUnsigned:=TRUE );
		MC_WriteParameter.Value:=16#0000;

		IF MC_WriteParameter.Done THEN
			MC_WriteParameter.Execute:=FALSE;
			iStep:=26;
		ELSIF NOT execute THEN
			iStep:=0;
		ELSIF MC_WriteParameter.Error THEN
			error:=TRUE;
		END_IF

	26:	//Read	0x3403:4	Motor (SM): Pole position encoder	49,5	°
		MC_ReadParameter.Enable:=TRUE;
		MC_ReadParameter.ParameterNumber:=L_MC1P_IndexToParameter2(
				uiIndex:=16#3403 ,
				usiSubIndex:=4 ,
				uiByteLength:=2 ,
				xUnsigned:=TRUE );

		IF MC_ReadParameter.Valid THEN
			polePositionNew:=MC_ReadParameter.Value;
			MC_ReadParameter.Enable:=FALSE;
			iStep:=28;
		ELSIF NOT execute THEN
			iStep:=0;
		ELSIF MC_ReadParameter.Error THEN
			error:=TRUE;
		END_IF

	28://Save	0x3403:4	Motor (SM): Pole position encoder	51,7	°
		MC_WriteParameter.Execute:=TRUE;
		MC_WriteParameter.ParameterNumber:=L_MC1P_IndexToParameter2(
				uiIndex:=16#3403 ,
				usiSubIndex:=4 ,
				uiByteLength:=2 ,
				xUnsigned:=TRUE );
		MC_WriteParameter.Value:=polePositionNew;

		IF MC_WriteParameter.Done THEN
			MC_WriteParameter.Execute:=FALSE;
			iStep:=30;
		ELSIF NOT execute THEN
			iStep:=0;
		ELSIF MC_WriteParameter.Error THEN
			error:=TRUE;
		END_IF

	30:	//Write	0x3025:0	Mode: Selection	CiA402 mode active [0]
		MC_WriteParameter.Execute:=TRUE;
		MC_WriteParameter.ParameterNumber:=L_MC1P_IndexToParameter2(
				uiIndex:=16#3025 ,
				usiSubIndex:=0 ,
				uiByteLength:=1 ,
				xUnsigned:=TRUE );
		MC_WriteParameter.Value:=0;

		IF MC_WriteParameter.Done THEN
			MC_WriteParameter.Execute:=FALSE;
			iStep:=32;
		ELSIF NOT execute THEN
			iStep:=0;
		ELSIF MC_WriteParameter.Error THEN
			error:=TRUE;
		END_IF

	32:	//Write	0x3024:0	Device control via PDO: Activation	Off [0]
		MC_WriteParameter.Execute:=TRUE;
		MC_WriteParameter.ParameterNumber:=L_MC1P_IndexToParameter2(
				uiIndex:=16#3024 ,
				usiSubIndex:=0 ,
				uiByteLength:=1 ,
				xUnsigned:=TRUE );
		MC_WriteParameter.Value:=1;

		IF MC_WriteParameter.Done THEN
			MC_WriteParameter.Execute:=FALSE;
			iStep:=100;
		ELSIF NOT execute THEN
			iStep:=0;
		ELSIF MC_WriteParameter.Error THEN
			error:=TRUE;
		END_IF

	100://Pole ident done
		done:=TRUE;
		doneOnce:=TRUE;
		busy:=FALSE;
		IF NOT execute THEN
			done:=FALSE;
			iStep:=0;
		END_IF
END_CASE

MC_WriteParameter(
	Axis:=ioAxis ,
	Execute:= ,
	ParameterNumber:= ,
	Value:= ,
	ExecutionMode:= ,
	Done=> ,
	Busy=> ,
	Error=> ,
	ErrorID=> );

MC_ReadParameter(
	Axis:=ioAxis ,
	Enable:= ,
	ParameterNumber:= ,
	Valid=> ,
	Busy=> ,
	Error=> ,
	ErrorID=> ,
	Value=> );

	(*
L_ETC_CoE_SdoRead4(
	xExecute:= ,
	xAbort:= ,
	usiCom:= ,
	uiDevice:=uiDevice ,
	wIndex:= ,
	bySubindex:= ,
	udiTimeOut:=100 ,
	xDone=> ,
	xBusy=> ,
	xError=> ,
	eErrorCode=> ,
	udiSdoAbort=> ,
	abyData=> ,
	szDataRead=> );

L_ETC_CoE_SdoWrite4(
	xExecute:= ,
	xAbort:= ,
	usiCom:= ,
	uiDevice:=uiDevice ,
	wIndex:= ,
	bySubindex:= ,
	udiTimeOut:=100 ,
	abyData:= ,
	usiDataLength:= ,
	xDone=> ,
	xBusy=> ,
	xError=> ,
	eErrorCode=> ,
	udiSdoAbort=> );
*)

END_FUNCTION_BLOCK

(* ---- L_SetIntQspRamp.pou ---- *)
FUNCTION_BLOCK L_SetIntQspRamp
VAR_IN_OUT
	Axis: AXIS_REF;
END_VAR
VAR_INPUT
	xExecute: BOOL;
	lrQspRamp: LREAL;
	lrQspTime: LREAL;
	xUseQspTime: BOOL;
END_VAR
VAR_OUTPUT
	xBusy: BOOL;
	xDone: BOOL;
	xError: BOOL;
	eErrorID: L_IE1P_Error;
END_VAR
VAR
	L_MC1P_ReadMachineData_Axis: L_MC1P_ReadMachineData;
	MC_WriteParameter_QspRamp: MC_WriteParameter;
	lrQspRamp_PosUnit: LREAL;
	RatedVel: LREAL;
	iStep: INT;
	uiIndexQspRamp: UINT;
	iSlotAxis: INT;
END_VAR

%LANGUAGE ST
//'L_SetIntQspRamp_i700'
//
//04.2016
//Lenze Vertrieb GmbH, Mirco Guddat

//Check if this is a i700 axis and witch slot
iSlotAxis:= L_GetSlot_i700(Axis:= Axis);

CASE iStep OF
	0: //Start
		xDone:= FALSE;
		xBusy:= FALSE;
		MC_WriteParameter_QspRamp.Execute:= FALSE;
		L_MC1P_ReadMachineData_Axis.xEnable:= FALSE;
		xError:= FALSE;
		eErrorID:= L_IE1P_Error.NoError;

		IF xExecute THEN
			iStep:= 10;
		END_IF

	10: //Read machine data
		xBusy:= TRUE;
		L_MC1P_ReadMachineData_Axis.xEnable:= TRUE;

		IF L_MC1P_ReadMachineData_Axis.xValid THEN
			iStep:= 20;
			ELSIF L_MC1P_ReadMachineData_Axis.xError THEN
				xError:= TRUE;
				eErrorID:= L_MC1P_ReadMachineData_Axis.eErrorID;
				iStep:= 40;
		END_IF

	20: //Calculate the internal quickstop ramp in Pos.Units/s2
		IF xUseQspTime THEN

			IF lrQspTime> 0 THEN
				IF (L_MC1P_ReadMachineData_Axis.lrFeedconstant= 0) OR (L_MC1P_ReadMachineData_Axis.dwGearDenominator= 0) THEN
					//Division by zero
					xError:= TRUE;
					lrQspRamp_PosUnit:= 16#7FFFFFFF;

					ELSE
						//The QSP-Time is calculated from rated velocity to standstill
						lrQspRamp_PosUnit:= ((L_MC1P_GetRatedVelocityAxis(Axis:= Axis)/ L_MC1P_ReadMachineData_Axis.lrFeedconstant) * (TO_LREAL(L_MC1P_ReadMachineData_Axis.dwGearNumerator) / TO_LREAL(L_MC1P_ReadMachineData_Axis.dwGearDenominator)) / lrQspTime) * 65536;
				END_IF

				ELSE
					//Zero dont work as QSP time, so we use the max. deceleration
					lrQspRamp_PosUnit:= 16#7FFFFFFF;
			END_IF

			ELSE
				IF lrQspRamp> 0.0 THEN
					IF (L_MC1P_ReadMachineData_Axis.lrFeedconstant= 0) OR (L_MC1P_ReadMachineData_Axis.dwGearDenominator= 0) THEN
						//Division by zero
						xError:= TRUE;
						lrQspRamp_PosUnit:= 16#7FFFFFFF;

						ELSE
							//Calculate QSP ramp
							lrQspRamp_PosUnit:= (lrQspRamp/ L_MC1P_ReadMachineData_Axis.lrFeedconstant) * (TO_LREAL(L_MC1P_ReadMachineData_Axis.dwGearNumerator) / TO_LREAL(L_MC1P_ReadMachineData_Axis.dwGearDenominator)) * 65536;
					END_IF

					ELSE
						//Zero dont work as QSP ramp, so we use the max. deceleration
						lrQspRamp_PosUnit:= 16#7FFFFFFF;
				END_IF
		END_IF

		iStep:= 30;

	30: //Write the parameter
		IF (iSlotAxis= 1) THEN
			uiIndexQspRamp:= 16#6085; //Index for slot 1
			ELSIF (iSlotAxis= 2) THEN
				uiIndexQspRamp:= 16#6885; //Index for slot 2
		END_IF

		MC_WriteParameter_QspRamp.Execute:= TRUE;

		IF MC_WriteParameter_QspRamp.Done THEN
			iStep:= 40;
			ELSIF MC_WriteParameter_QspRamp.Error THEN
				xError:= TRUE;
				eErrorID:= MC_WriteParameter_QspRamp.ErrorID;
		END_IF

	40: //finish
		xDone:= TRUE;
		xBusy:= FALSE;
		IF NOT xExecute THEN
			iStep:= 0;
		END_IF

END_CASE

L_MC1P_ReadMachineData_Axis(
	Axis:= Axis,
	xEnable:= ,
	xValid=> ,
	xBusy=> ,
	xError=> ,
	eErrorID=> ,
	lrFeedconstant=> ,
	dwGearDenominator=> ,
	dwGearNumerator=> ,
	dwPosResolution=> ,
	xOrientation=> ,
	eTraversingRange=> ,
	lrCycleLength=> ,
	xVirtual=> );

MC_WriteParameter_QspRamp(
	Axis:= Axis,
	Execute:= ,
	ParameterNumber:= L_MC1P_IndexToParameter(uiIndex:= uiIndexQspRamp, usiSubIndex:= 0, uiByteLength:= 4),
	Value:= lrQspRamp_PosUnit,
	ExecutionMode:= ,
	Done=> ,
	Busy=> ,
	Error=> ,
	ErrorID=> );

END_FUNCTION_BLOCK

(* ---- VirtualMaster.pou ---- *)
FUNCTION_BLOCK VirtualMaster
//Dataexchange CONTROL ===========
VAR_IN_OUT
	ioDataExchange					:  sUDT_VirtualMasterComm_Drive;
END_VAR
VAR_INPUT
	i_xPositionIsRetain				: BOOL;
	i_lrWindowStandstill			: LREAL;
	i_lrJogVel						: LREAL;
	i_VelMax						: LREAL;
END_VAR
VAR_OUTPUT
END_VAR
VAR
	//ControlWord
	internalControl					:	BOOL;
	Control_Local			 		:	sUDT_VirtualMasterComm_Drive_Control;			//output to plc

	//StatusWord

	//instance
	AxisControl						: L_TF2P_VirtualMasterBase;
	SetTorqueError					: L_IE1P_SetErrorSingle;
END_VAR
VAR_IN_OUT
	ioSlaveAxis						: AXIS_REF;
END_VAR
VAR RETAIN PERSISTENT
	lrRetainPosition				: LREAL;
END_VAR

%LANGUAGE ST

ReadInputs();
VirtualMasterParameters();
VirtualMaster();
SetTorqueLimits();
BrakeLogic();
WriteOutputs();

lrRetainPosition:=ioSlaveAxis.lrSetPosition;

END_FUNCTION_BLOCK

METHOD BrakeLogic
VAR_INPUT

END_VAR
VAR_INST
	BrakeInterface			: L_MC1P_BrakeInterface;
END_VAR

VAR

END_VAR
%LANGUAGE ST

BrakeInterface(
	Axis:= ioSlaveAxis,
	xEnable:= NOT ioSlaveAxis.xVirtual ,
	xReleaseBrake:= Control_Local.ReleaseBrake,
	lrTorqueAdd:= ,
	xBrakeModeActivate:= ,
	eBrakeMode:= ,
	xValid=> ,
	xBusy=> ,
	xError=> ,
	eErrorID=> ,
	xBrakeReleaseOut=> ,
	xBrakeReleased=> ,
	lrActTorque=> ,
	lrStartingTorqueSaved=> ,
	lrStartingTorqueEffective=> ,
	eBrakeModeActive=> );
END_METHOD

METHOD ReadInputs
VAR_INPUT
END_VAR

%LANGUAGE ST

//activate internal control
IF NOT internalControl THEN
	Control_Local	:= ioDataExchange.Control;
END_IF

END_METHOD

METHOD SetTorqueLimits
VAR_INPUT

END_VAR
VAR_INST
	TorqueLimit						: L_MC1P_SetTorqueLimit;
	lrRefTorqueAxis					: LREAL;
	lrActTorqueProcent				: LREAL;
	ResetError						: L_IE1P_ResetError;
END_VAR

VAR

END_VAR
%LANGUAGE ST

//Max torque on the axis. If the machine doesn't stop due to a programming error, this part ensures that the torque never gets too high.
TorqueLimit(
	Axis:= ioSlaveAxis,
	xEnable:= NOT ioSlaveAxis.xVirtual ,
	xSetTorqueLimitPos:= TRUE,
	lrTorqueLimitPos:= (Control_Local.TorqueLimit/100)*1.1, 				//The max torque allowed on the axis is 10% higher then the alarm value.
	xSetTorqueLimitNeg:= TRUE,
	lrTorqueLimitNeg:= (Control_Local.TorqueLimit/100)*1.1, 				//The max torque allowed on the axis is 10% higher then the alarm value.
	xTorqueInputAsPercent:= TRUE,
	xBusy=> ,
	xError=> ,
	eErrorID=> );

lrRefTorqueAxis := L_MC1P_GetRatedTorqueAxis(Axis:=ioSlaveAxis);
//Torque limit error
IF lrRefTorqueAxis > 0 THEN
	lrActTorqueProcent := ABS(ioSlaveAxis.lrActTorque/lrRefTorqueAxis);
END_IF

SetTorqueError(
	ModuleHandler:= ,
	ErrorHandler:=ioSlaveAxis ,
	xSetError:=lrActTorqueProcent > (Control_Local.TorqueLimit/100) ,
	eSeverity:=L_IE1P_SeverityLevel.Fault_Qsp_Cinh ,
	wTextRefId:= ATD_Errorlist,
	wErrorId:= 1,
	eReaction:= ,
	eGroup:= ,
	xError=> ,
	eErrorID=> ,
	scErrorInformation=> );

ResetError(
	ModuleHandler:= ,
	ErrorHandler:=ioSlaveAxis ,
	xResetError:=AxisControl.xResetError ,
	xError=> ,
	eErrorID=> ,
	xErrorResetActive=> ,
	xResetActive=> );
END_METHOD

METHOD VirtualMaster
VAR_INPUT
END_VAR
VAR_INST

END_VAR
VAR_INST
	MC_SetPosition:MC_SetPosition;
	SetIntQspRamp			: L_SetIntQspRamp;
	lrDecErrorStopOld		: LREAL;
END_VAR
%LANGUAGE ST

AxisControl.scCtrlBasicMotion.xResetHomePosition:=Control_Local.ResetHomePos;

AxisControl(
	xEnable:=TRUE ,
	xEnableOperation:= Control_Local.Enable,
	xResetError:=Control_Local.ResetError ,
	xQSPApplication:= ,
	xAbort:=NOT Control_Local.StartMovement ,
	xJogPos:= ,
	xJogNeg:= ,
	xHomeExecute:= Control_Local.SetHomePos,
	lrOverride:= ,
	scCtrlBasicMotion:= ,
	scPar:= ,
	Axis:=ioSlaveAxis ,
	scAccessPoints:= ,
	MasterValues:= ,
	xContinuous:=(Control_Local.StartMovement AND (NOT AxisControl.xAbortBusy)),
	xCycleExecute:= ,
	xLoadStartPos:= ,
	lrSetVel:= ,
	xSyncIn:= ,
	xReadyForOperation=> ,
	xOperationEnabled=> ,
	xReadyForMotion=> ,
	xError=> ,
	xWarning=> ,
	eErrorID=> ,
	xSTOActive=> ,
	xQSPActive=> ,
	xAbortBusy=> ,
	xAbortDone=> ,
	xJoggingBusy=> ,
	xHomingBusy=> ,
	xHomingDone=> ,
	xIsHomed=> ,
	eTMState=> ,
	scStatusBasicMotion=> ,
	lrActVel=> ,
	lrSetVelOut=> ,
	lrActPos=> ,
	lrSetPosOut=> ,
	lrActFollowingError=> ,
	xContinuousMotionBusy=> ,
	xCyclicMotionBusy=> ,
	xCyclicMotionDone=> ,
	xMoveToTargetPosBusy=> ,
	xMoveToTargetPosDone=> ,
	xInTarget=> ,
	xAccDecSync=> ,
	xSynchronised=> );

MC_SetPosition(
	Axis:=ioSlaveAxis ,
	Execute:=i_xPositionIsRetain AND ioSlaveAxis.xAxisAvailable ,
	Position:=lrRetainPosition ,
	Relative:= ,
	ExecutionMode:= ,
	RestartPositioning:= ,
	UseSettingsFromHomingMode:= ,
	Done=> ,
	Busy=> ,
	Error=> ,
	ErrorID=> );

SetIntQspRamp(
	Axis:=ioSlaveAxis ,
	xExecute:=ioSlaveAxis.xAxisAvailable AND NOT ioSlaveAxis.xVirtual AND (lrDecErrorStopOld=ioSlaveAxis.lrDecErrorStop) ,
	lrQspRamp:=ioSlaveAxis.lrDecErrorStop ,
	lrQspTime:= ,
	xUseQspTime:= ,
	xBusy=> ,
	xDone=> ,
	xError=> ,
	eErrorID=> );
lrDecErrorStopOld:=ioSlaveAxis.lrDecErrorStop;
END_METHOD

METHOD VirtualMasterParameters
VAR_INPUT
END_VAR

%LANGUAGE ST
//General
//ioSlaveAxis.scPar.WindowStandStill:=i_lrWindowStandstill;
//ioSlaveAxis.scPar.JoggingSetVel:=i_lrJogVel;
//ioSlaveAxis.scPar.JoggingSetAcc:=i_lrJogVel*10;
//ioSlaveAxis.scPar.JoggingSetDec:=i_lrJogVel*10;
//ioSlaveAxis.scPar.JoggingSetJerk:=0;

IF (Control_Local.VelUnit>i_VelMax) THEN
	AxisControl.lrSetVel:=i_VelMax;
ELSE
	AxisControl.lrSetVel:=Control_Local.VelUnit;
END_IF

AxisControl.scPar.eDirection:=MC_DIRECTION.mcPositiveDirection;
AxisControl.scPar.lrVel:=Control_Local.VelUnit;
AxisControl.scPar.lrAcc:=Control_Local.AccUnit;
AxisControl.scPar.lrDec:=Control_Local.DecUnit;
AxisControl.scPar.lrJerk:=0;
AxisControl.scPar.lrTargetPos:=Control_Local.PosUnit;

//Sync with external encoder NOT USED
AxisControl.scPar.lrSyncVel:=5;
AxisControl.scPar.lrSyncAcc:=10;
AxisControl.scPar.lrSyncDec:=10;
AxisControl.scPar.lrSyncJerk:=0;
AxisControl.scPar.lrStartPos:=0;

END_METHOD

METHOD WriteOutputs
VAR_INPUT
END_VAR
VAR_INST

END_VAR

%LANGUAGE ST

ioDataExchange.Status.DriveCommAlive				:= ioSlaveAxis.xCommunicationOK;
ioDataExchange.Status.ReadyForOperation				:= AxisControl.xReadyForOperation;
ioDataExchange.Status.ReadyForMotion				:= AxisControl.xReadyForMotion;
ioDataExchange.Status.HomingPosOK					:= AxisControl.xIsHomed;
ioDataExchange.Status.InPosition					;//writen in statemachine
ioDataExchange.Status.VelocitySetpointReached		;//writen in statemachine
ioDataExchange.Status.ActSpeed						:= AxisControl.lrActVel;
ioDataExchange.Status.ActPos						:= AxisControl.lrActPos;

END_METHOD
